Fanuc TP program (LS listing): ZZZ9_BAK2.LS

/PROG  ZZZ9_BAK2
/ATTR
OWNER		= KAREL;
COMMENT		= "";
PROG_SIZE	= 132;
CREATE		= DATE 21-03-23  TIME 17:19:50;
MODIFIED	= DATE 21-03-23  TIME 17:19:50;
FILE_NAME	= ;
VERSION		= 0;
LINE_COUNT	= 0;
MEMORY_SIZE	= 376;
PROTECT		= READ_WRITE;
TCD:  STACK_SIZE	= 0,
      TASK_PRIORITY	= 50,
      TIME_SLICE	= 0,
      BUSY_LAMP_OFF	= 0,
      ABORT_REQUEST	= 0,
      PAUSE_REQUEST	= 0;
DEFAULT_GROUP	= 1,*,*,*,*;
CONTROL_CODE	= 00000000 00000000;
/APPL
/MN
/POS
/END
